Fanuc KAREL source: kb00153.KL

-- PROVISIONAL review KL for V770-1; original PC SHA256 99bbab02688c3893f70f7a2e40b574191d667efddfb836ad4a8dae245ffcc349
-- Incomplete behavior may be omitted. Consult companion uncertainty JSON. Do not deploy.
PROGRAM KB00153
%NOLOCKGROUP
BEGIN
  -- UNRESOLVED_PC offsets 5-14; opcodes 3F,75
  -- UNRESOLVED_PC offsets 19-26; opcodes 9D,23
  -- UNRESOLVED_PC offsets 31-38; opcodes 9D,23
  -- UNRESOLVED_PC offsets 43-50; opcodes 9D,23
  -- UNRESOLVED_PC offsets 55-62; opcodes 9D,23
  -- UNRESOLVED_PC offsets 67-74; opcodes 9D,23
  -- UNRESOLVED_PC offsets 79-121; opcodes 27,22,2A,22,22,22,22,22,31
  -- UNRESOLVED_PC offsets 126-130; opcodes 7F
END KB00153
